Universal Robots PolyScope program: advanced_template.urp

ProgramRoot setBeforeStartSequence=true; setInitialVariableValues=true; directory=/programs/robotiq_2f_gripper_programs; kinematics=(a=[0, -0.425, -0.39225, 0, 0, 0], d=[0.08916, 0, 0, 0.10915, 0.09465, 0.0823], alpha=[1.5708, 0, 0, 1.5708, -1.5708, 0], deltaTheta=[0, 0, 0, 0, 0, 0], status=notInitialized); name=advanced_template; robotEnvironmentFileName=default; serialNumberRobot=2013212154
  InitVariables 
  BeforeStart description=COMMAND_SEQUENCE_BEFORE_PROGRAM_START; name=BeforeStart
    Script type=1; scriptFile=/programs/robotiq_2f_gripper_programs/rq_before_start.script
    Script type=1; scriptFile=/programs/robotiq_2f_gripper_programs/rq_script.script
    CallSubProgram subProgramNodeToCall=rq_print_driver_version()
    Assignment assignmentValueSource=0; expr=0; operatorValueType=INTEGER; valueSource=EXPRESSION; variable=0
    Assignment assignmentValueSource=0; expr=0; operatorValueType=INTEGER; valueSource=EXPRESSION; variable=0
    Assignment assignmentValueSource=0; expr=0; operatorValueType=INTEGER; valueSource=EXPRESSION; variable=0
    Assignment assignmentValueSource=0; expr=0; operatorValueType=INTEGER; valueSource=EXPRESSION; variable=0
    Assignment assignmentValueSource=0; expr=255; operatorValueType=INTEGER; valueSource=EXPRESSION; variable=255
    Assignment assignmentValueSource=0; expr=255; operatorValueType=INTEGER; valueSource=EXPRESSION; variable=255
  MainProgram cartesianAcceleration=1.2; cartesianSpeed=0.25; jointAcceleration=1.3962634015954636; jointSpeed=1.0471975511965976; moveAsFastAsPossible=true; sharedProcessMoveBlendRadius=0.025; featureReference=(installationNameReference=Base); motionType=JOINT_SPACE
    CallSubProgram subProgramNodeToCall=rq_activate_and_wait()
    While count=0; type=LOOP_FOREVER
      CallSubProgram subProgramNodeToCall=rq_close_and_wait()
      CallSubProgram subProgramNodeToCall=rq_open_and_wait()
  SubProgram [hidden by the author, left out]
  subProgramToCall [hidden by the author, left out]
  SubProgram [hidden by the author, left out]
  SubProgram [hidden by the author, left out]
  SubProgram [hidden by the author, left out]
  subProgramToCall [hidden by the author, left out]
  SubProgram [hidden by the author, left out]
  SubProgram [hidden by the author, left out]
  SubProgram [hidden by the author, left out]
  SubProgram [hidden by the author, left out]
  SubProgram [hidden by the author, left out]
  SubProgram [hidden by the author, left out]
  SubProgram [hidden by the author, left out]
  subProgramToCall [hidden by the author, left out]
  SubProgram [hidden by the author, left out]
  SubProgram [hidden by the author, left out]
  SubProgram [hidden by the author, left out]
  SubProgram [hidden by the author, left out]
  SubProgram [hidden by the author, left out]
  SubProgram [hidden by the author, left out]
  SubProgram [hidden by the author, left out]
  SubProgram [hidden by the author, left out]
  SubProgram [hidden by the author, left out]
  SubProgram [hidden by the author, left out]
  subProgramToCall [hidden by the author, left out]
  SubProgram [hidden by the author, left out]
  SubProgram [hidden by the author, left out]
  SubProgram [hidden by the author, left out]
  SubProgram [hidden by the author, left out]
  SubProgram [hidden by the author, left out]
  SubProgram [hidden by the author, left out]
